//{attribute 'pack_mode' := '8'}
TYPE ST_HierarchyDataList :
STRUCT

	TrackingLevels		:STRING(13);
	HierarchyDataPK	:ST_HierarchyData;
	HierarchyDataOUT	:ST_HierarchyData;
	HierarchyDataCS	:ST_HierarchyData;
	HierarchyDataPAL	:ST_HierarchyData;
END_STRUCT
END_TYPE

(* stored: Version 1.1.0.1
   DUT ST_HierarchyDataList: Id {0b02b9ba-c034-46f0-a487-a20edab0b3b9} *)
